FUNCTION_BLOCK CompositeTestBlock2
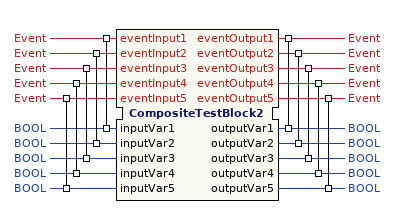
  EVENT_INPUT
    eventInput1 WITH inputVar1;
    eventInput2 WITH inputVar2;
    eventInput3 WITH inputVar3;
    eventInput4 WITH inputVar4;
    eventInput5 WITH inputVar5;
  END_EVENT
  EVENT_OUTPUT
    eventOutput1 WITH outputVar1;
    eventOutput2 WITH outputVar2;
    eventOutput3 WITH outputVar3;
    eventOutput4 WITH outputVar4;
    eventOutput5 WITH outputVar5;
  END_EVENT
  VAR_INPUT
    inputVar1 : BOOL;
    inputVar2 : BOOL;
    inputVar3 : BOOL;
    inputVar4 : BOOL;
    inputVar5 : BOOL;
  END_VAR
  VAR_OUTPUT
    outputVar1 : BOOL;
    outputVar2 : BOOL;
    outputVar3 : BOOL;
    outputVar4 : BOOL;
    outputVar5 : BOOL;
  END_VAR
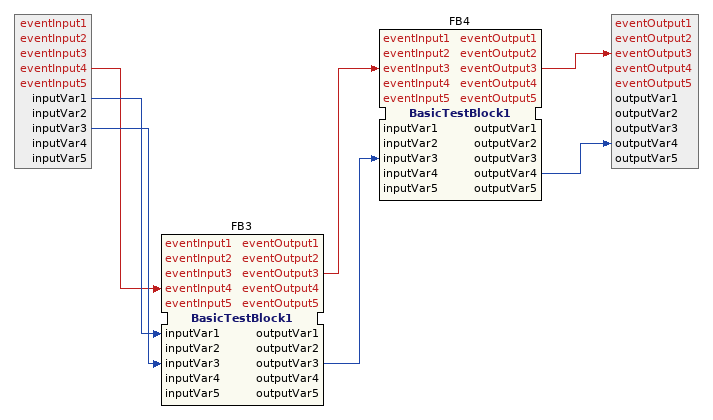
  FBS
    FB3 : BasicTestBlock1;
    FB4 : BasicTestBlock1;
  END_FBS
  EVENT_CONNECTIONS
    FB3.eventOutput3 TO FB4.eventInput3;
    FB4.eventOutput3 TO eventOutput3;
    eventInput4 TO FB3.eventInput4;
  END_CONNECTIONS
  DATA_CONNECTIONS
    FB3.outputVar3 TO FB4.inputVar3;
    FB4.outputVar4 TO outputVar4;
    inputVar1 TO FB3.inputVar1;
    inputVar3 TO FB3.inputVar3;
  END_CONNECTIONS
END_FUNCTION_BLOCK
